% RSLogix 500 project Servodriver_Application.RSS, saved by version 8.30.00.16 %
PROJECT "UNTITLED"    % processor: Bul.1763 MicroLogix 1100 Series B %

PROGRAM FILES
  LAD 2 "MAIN"  6 rungs
  LAD 3 "DIGITAL_IO"  7 rungs
  LAD 4 "CYCLE_STAT"  7 rungs
  LAD 5 "CONTROL"  10 rungs

DATA FILES
  O0 OUTPUT  4 elements
  I1 INPUT  6 elements
  S2 STATUS  66 elements
  B3 BINARY  2 elements
  T4 TIMER  3 elements
  C5 COUNTER  1 elements
  R6 CONTROL  1 elements
  N7 INTEGER  1 elements
  F8 FLOAT  1 elements

LADDER 2 "MAIN"
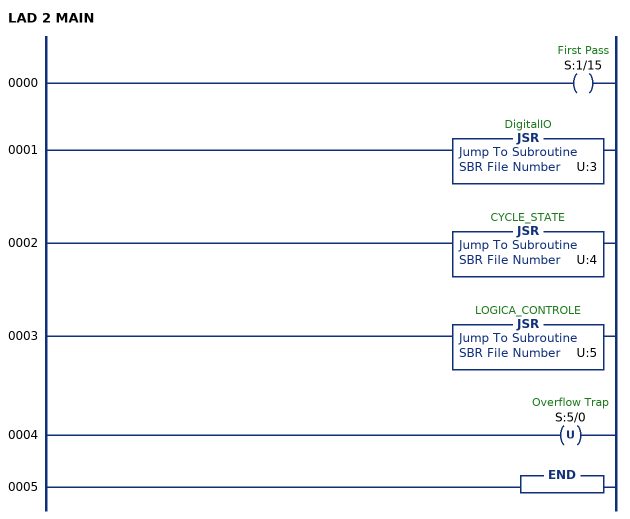
% Rung: 0 %
SOR OTE S:1/15 EOR
%   S:1/15  "First Pass" %
% Rung: 1 %
SOR JSR U:3 EOR
%   U:3  "DigitalIO" %
% Rung: 2 %
SOR JSR U:4 EOR
%   U:4  "CYCLE_STATE" %
% Rung: 3 %
SOR JSR U:5 EOR
%   U:5  "LOGICA_CONTROLE" %
% Rung: 4 %
SOR OTU S:5/0 EOR
%   S:5/0  "Overflow Trap" %
% Rung: 5 %
SOR END EOR

LADDER 3 "DIGITAL_IO"
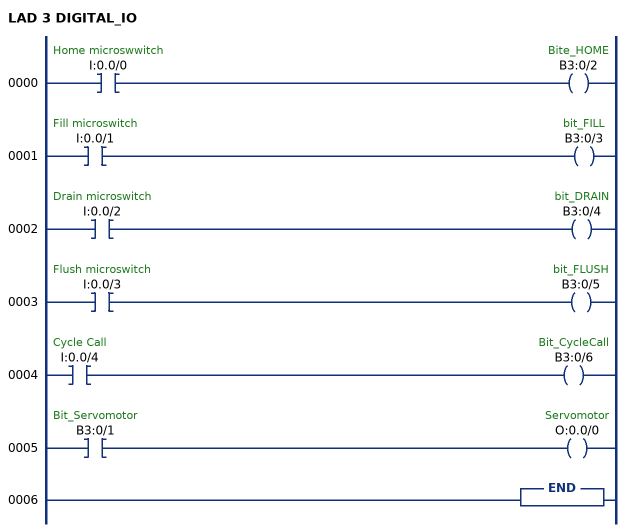
% Rung: 0 %
SOR XIC I:0.0/0 OTE B3:0/2 EOR
%   I:0.0/0  "Home microswwitch" %
%   B3:0/2  "Bite_HOME" %
% Rung: 1 %
SOR XIC I:0.0/1 OTE B3:0/3 EOR
%   I:0.0/1  "Fill microswitch" %
%   B3:0/3  "bit_FILL" %
% Rung: 2 %
SOR XIC I:0.0/2 OTE B3:0/4 EOR
%   I:0.0/2  "Drain microswitch" %
%   B3:0/4  "bit_DRAIN" %
% Rung: 3 %
SOR XIC I:0.0/3 OTE B3:0/5 EOR
%   I:0.0/3  "Flush microswitch" %
%   B3:0/5  "bit_FLUSH" %
% Rung: 4 %
SOR XIC I:0.0/4 OTE B3:0/6 EOR
%   I:0.0/4  "Cycle Call" %
%   B3:0/6  "Bit_CycleCall" %
% Rung: 5 %
SOR XIC B3:0/1 OTE O:0.0/0 EOR
%   B3:0/1  "Bit_Servomotor" %
%   O:0.0/0  "Servomotor" %
% Rung: 6 %
SOR END EOR

LADDER 4 "CYCLE_STAT"
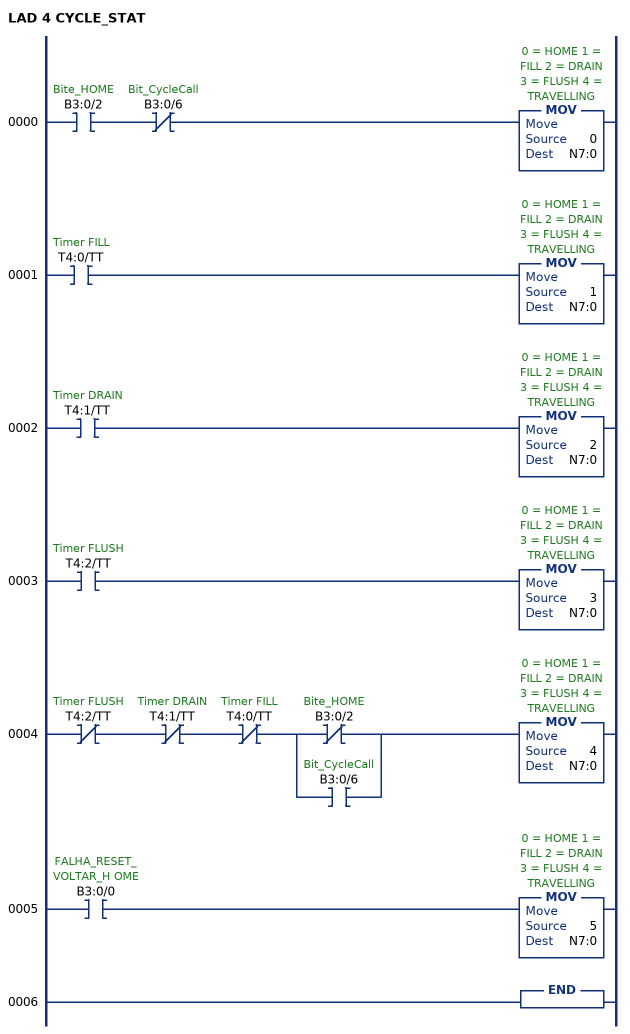
% Rung: 0 %
SOR XIC B3:0/2 XIO B3:0/6 MOV 0 N7:0 EOR
%   B3:0/2  "Bite_HOME" %
%   B3:0/6  "Bit_CycleCall" %
%   N7:0  "0 = HOME 1 = FILL 2 = DRAIN 3 = FLUSH 4 = TRAVELLING" %
% Rung: 1 %
SOR XIC T4:0/TT MOV 1 N7:0 EOR
%   T4:0  "Timer FILL" %
%   N7:0  "0 = HOME 1 = FILL 2 = DRAIN 3 = FLUSH 4 = TRAVELLING" %
% Rung: 2 %
SOR XIC T4:1/TT MOV 2 N7:0 EOR
%   T4:1  "Timer DRAIN" %
%   N7:0  "0 = HOME 1 = FILL 2 = DRAIN 3 = FLUSH 4 = TRAVELLING" %
% Rung: 3 %
SOR XIC T4:2/TT MOV 3 N7:0 EOR
%   T4:2  "Timer FLUSH" %
%   N7:0  "0 = HOME 1 = FILL 2 = DRAIN 3 = FLUSH 4 = TRAVELLING" %
% Rung: 4 %
SOR XIO T4:2/TT XIO T4:1/TT XIO T4:0/TT BST XIO B3:0/2 NXB XIC B3:0/6 BND MOV 4 N7:0 EOR
%   T4:2  "Timer FLUSH" %
%   T4:1  "Timer DRAIN" %
%   T4:0  "Timer FILL" %
%   B3:0/2  "Bite_HOME" %
%   B3:0/6  "Bit_CycleCall" %
%   N7:0  "0 = HOME 1 = FILL 2 = DRAIN 3 = FLUSH 4 = TRAVELLING" %
% Rung: 5 %
SOR XIC B3:0/0 MOV 5 N7:0 EOR
%   B3:0/0  "FALHA_RESET_VOLTAR_H OME" %
%   N7:0  "0 = HOME 1 = FILL 2 = DRAIN 3 = FLUSH 4 = TRAVELLING" %
% Rung: 6 %
SOR END EOR

LADDER 5 "CONTROL"
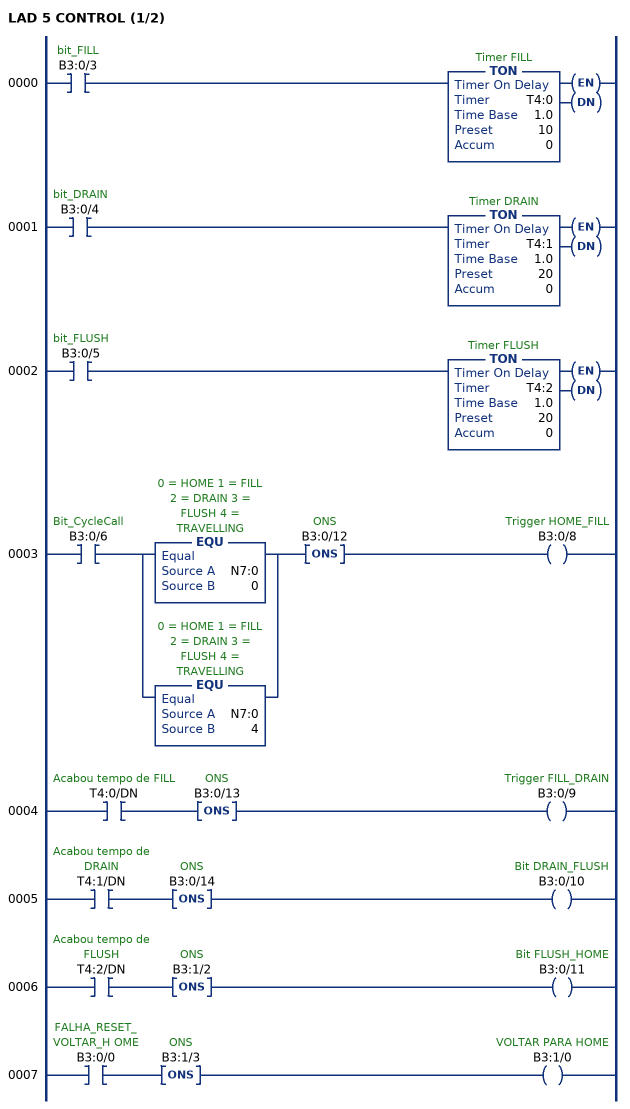
% Rung: 0 %
SOR XIC B3:0/3 TON T4:0 1.0 10 0 EOR
%   B3:0/3  "bit_FILL" %
%   T4:0  "Timer FILL" %
% Rung: 1 %
SOR XIC B3:0/4 TON T4:1 1.0 20 0 EOR
%   B3:0/4  "bit_DRAIN" %
%   T4:1  "Timer DRAIN" %
% Rung: 2 %
SOR XIC B3:0/5 TON T4:2 1.0 20 0 EOR
%   B3:0/5  "bit_FLUSH" %
%   T4:2  "Timer FLUSH" %
% Rung: 3 %
SOR XIC B3:0/6 BST EQU N7:0 0 NXB EQU N7:0 4 BND ONS B3:0/12 OTE B3:0/8 EOR
%   B3:0/6  "Bit_CycleCall" %
%   N7:0  "0 = HOME 1 = FILL 2 = DRAIN 3 = FLUSH 4 = TRAVELLING" %
%   B3:0/12  "ONS" %
%   B3:0/8  "Trigger HOME_FILL" %
% Rung: 4 %
SOR XIC T4:0/DN ONS B3:0/13 OTE B3:0/9 EOR
%   T4:0/DN  "Acabou tempo de FILL" %
%   B3:0/13  "ONS" %
%   B3:0/9  "Trigger FILL_DRAIN" %
% Rung: 5 %
SOR XIC T4:1/DN ONS B3:0/14 OTE B3:0/10 EOR
%   T4:1/DN  "Acabou tempo de DRAIN" %
%   B3:0/14  "ONS" %
%   B3:0/10  "Bit DRAIN_FLUSH" %
% Rung: 6 %
SOR XIC T4:2/DN ONS B3:1/2 OTE B3:0/11 EOR
%   T4:2/DN  "Acabou tempo de FLUSH" %
%   B3:1/2  "ONS" %
%   B3:0/11  "Bit FLUSH_HOME" %
% Rung: 7 %
SOR XIC B3:0/0 ONS B3:1/3 OTE B3:1/0 EOR
%   B3:0/0  "FALHA_RESET_VOLTAR_H OME" %
%   B3:1/3  "ONS" %
%   B3:1/0  "VOLTAR PARA HOME" %

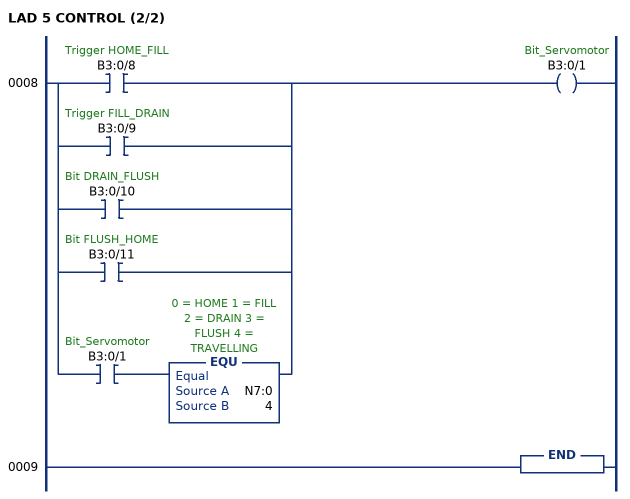
% Rung: 8 %
SOR BST XIC B3:0/8 NXB XIC B3:0/9 NXB XIC B3:0/10 NXB XIC B3:0/11 NXB XIC B3:0/1 EQU N7:0 4 BND OTE B3:0/1 EOR
%   B3:0/8  "Trigger HOME_FILL" %
%   B3:0/9  "Trigger FILL_DRAIN" %
%   B3:0/10  "Bit DRAIN_FLUSH" %
%   B3:0/11  "Bit FLUSH_HOME" %
%   B3:0/1  "Bit_Servomotor" %
%   N7:0  "0 = HOME 1 = FILL 2 = DRAIN 3 = FLUSH 4 = TRAVELLING" %
% Rung: 9 %
SOR END EOR

OTHER DOCUMENTED ADDRESSES
  B3:0/7  "Trigger HOME_FILL"

DATA TABLE (non-zero values as saved)
DATA B3
% B3:0 % 0X1046 0X0000
DATA T4
% .PRE .ACC %
% T4:0 % 10 0
% T4:1 % 20 0
% T4:2 % 20 0
DATA N7
% N7:0 % 4
